// TIA Portal project "Teste_Elipse" (V17)

(* hardware
DEVICE "S7-1200 station_1"  S7-1200 Station
   slot 0: "Rack_0"  S7-1200 Rack  Rack  V1.0
   slot 1: "PLC_1"  CPU 1214C DC/DC/DC  6ES7 214-1AG31-0XB0  V3.0
*)

// ===== PLC "PLC_1"  CPU 1214C DC/DC/DC =====

VAR_GLOBAL   // PLC tag table "Default tag table"
   "Clock_Byte" AT %MB5 : Byte;
   "Clock_10Hz" AT %M5.0 : Bool;
   "Clock_5Hz" AT %M5.1 : Bool;
   "Clock_2.5Hz" AT %M5.2 : Bool;
   "Clock_2Hz" AT %M5.3 : Bool;
   "Clock_1.25Hz" AT %M5.4 : Bool;
   "Clock_1Hz" AT %M5.5 : Bool;
   "Clock_0.625Hz" AT %M5.6 : Bool;
   "Clock_0.5Hz" AT %M5.7 : Bool;
   "Carrega" AT %M0.0 : Bool;
   "Descarregar" AT %M0.1 : Bool;
   "Carregando" AT %M0.2 : Bool;
   "Descarregando" AT %M0.3 : Bool;
   "Ligar" AT %I0.0 : Bool;
   "Desligar" AT %I0.1 : Bool;
   "LEDCarga" AT %Q0.0 : Bool;
   "LEDDescarga" AT %Q0.1 : Bool;
   "MEM_Carregado" AT %M0.4 : Bool;
   "MEM_Descarregado" AT %M0.5 : Bool;
END_VAR

DATA_BLOCK "Data_block_1"   // DB2
{ S7_Optimized_Access := 'FALSE' }
VERSION : 0.1
   VAR
      Ligar : Bool;
      Desligar : Bool;
   END_VAR
BEGIN
END_DATA_BLOCK

// folder: System blocks/Program resources

DATA_BLOCK "IEC_Counter_0_DB"   // DB1
{ S7_Optimized_Access := 'TRUE' }
AUTHOR : Simatic
FAMILY : IEC
NAME : CNTR
VERSION : 1.0
// stored: InstanceOfName IEC_COUNTER
"IEC_COUNTER"
BEGIN
END_DATA_BLOCK

// folder: (top level)

ORGANIZATION_BLOCK "Main"   // OB1, LAD, ProgramCycle
TITLE = "Main Program Sweep (Cycle)"
{ S7_Optimized_Access := 'TRUE' }
VERSION : 0.1
BEGIN

REGION Network 1
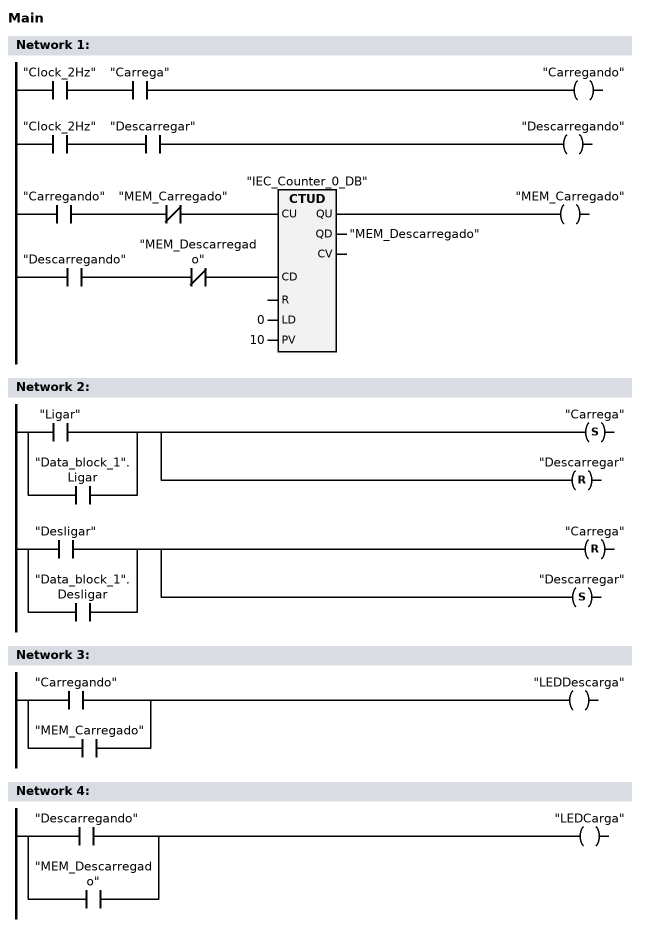
   "Carregando" := "Clock_2Hz" AND "Carrega";
   "Descarregando" := "Clock_2Hz" AND "Descarregar";
   "IEC_Counter_0_DB".CTUD(CU := "Carregando" AND NOT "MEM_Carregado",
                           CD := "Descarregando" AND NOT "MEM_Descarregado",
                           LD := 0,
                           PV := 10,
                           QD => "MEM_Descarregado");
   "MEM_Carregado" := "IEC_Counter_0_DB".QU;
END_REGION

REGION Network 2
   RUNG wire#powerrail
      Contact( "Ligar" )
      wire#w1
      S_Coil( "Carrega" )
   END_RUNG
   RUNG wire#powerrail
      Contact( "Data_block_1".Ligar )
   END_RUNG wire#w1
   RUNG wire#w1
      R_Coil( "Descarregar" )
   END_RUNG
   RUNG wire#powerrail
      Contact( "Desligar" )
      wire#w2
      R_Coil( "Carrega" )
   END_RUNG
   RUNG wire#powerrail
      Contact( "Data_block_1".Desligar )
   END_RUNG wire#w2
   RUNG wire#w2
      S_Coil( "Descarregar" )
   END_RUNG
   // the same network as SCL:
   IF "Ligar" OR "Data_block_1".Ligar THEN
       "Carrega" := TRUE;
       "Descarregar" := FALSE;
   END_IF;
   IF "Desligar" OR "Data_block_1".Desligar THEN
       "Carrega" := FALSE;
       "Descarregar" := TRUE;
   END_IF;
END_REGION

REGION Network 3
   RUNG wire#powerrail
      Contact( "Carregando" )
      wire#w1
      Coil( "LEDDescarga" )
   END_RUNG
   RUNG wire#powerrail
      Contact( "MEM_Carregado" )
   END_RUNG wire#w1
   // the same network as SCL:
   "LEDDescarga" := "Carregando" OR "MEM_Carregado";
END_REGION

REGION Network 4
   RUNG wire#powerrail
      Contact( "Descarregando" )
      wire#w1
      Coil( "LEDCarga" )
   END_RUNG
   RUNG wire#powerrail
      Contact( "MEM_Descarregado" )
   END_RUNG wire#w1
   // the same network as SCL:
   "LEDCarga" := "Descarregando" OR "MEM_Descarregado";
END_REGION
END_ORGANIZATION_BLOCK